TYPE "HU_Pump_Par"
VERSION : 0.1
// Block: HU_Pump_Par
   STRUCT
      DelayCheckFilterClogged : Time;
      DelayPumpInactivity : Time;
      DelayEvPressureStart : Time;
      DelayEvPressureStop : Time;
      DelayPressureRunning : Time;
   END_STRUCT;

END_TYPE
